FUNCTION_BLOCK StackControlLogic (* Basic Function Block Type *)
  (* Standard: 61499-2 *)
  (* Version 0.0, 9/26/2018, dmidro, nxtControl GmbH, Template *)
  PACKAGE Main;
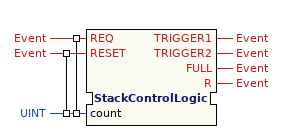
  EVENT_INPUT
    REQ WITH count; (* Normal Execution Request *)
    RESET WITH count;
  END_EVENT
  EVENT_OUTPUT
    TRIGGER1; (* Execution Confirmation *)
    TRIGGER2;
    FULL;
    R;
  END_EVENT
  VAR_INPUT
    count : UINT;
  END_VAR
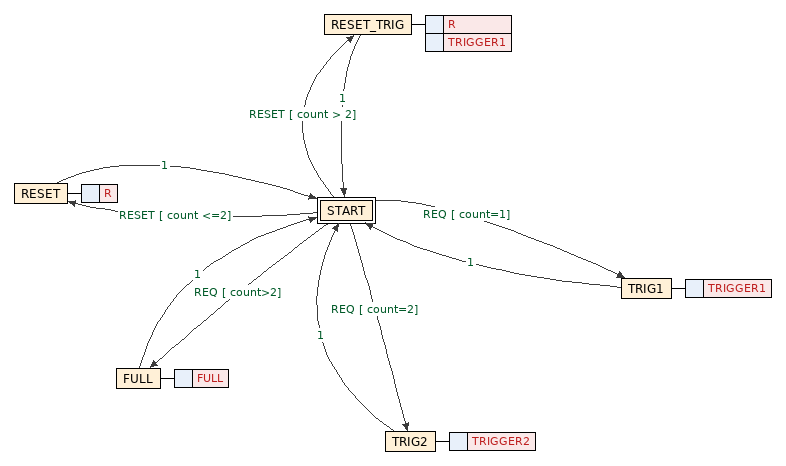
  EC_STATES
    START; (* Initial State *)
    TRIG1 : -> TRIGGER1; (* Normal execution *)
    TRIG2 : -> TRIGGER2;
    FULL : -> FULL;
    RESET : -> R;
    RESET_TRIG : -> R, -> TRIGGER1;
  END_STATES
  EC_TRANSITIONS
    START TO TRIG1 := REQ [ count=1];
    START TO TRIG2 := REQ [ count=2];
    TRIG2 TO START := 1;
    START TO FULL := REQ [ count>2];
    FULL TO START := 1;
    TRIG1 TO START := 1;
    START TO RESET := RESET [ count <=2];
    RESET TO START := 1;
    START TO RESET_TRIG := RESET [ count > 2];
    RESET_TRIG TO START := 1;
  END_TRANSITIONS
END_FUNCTION_BLOCK
